// TIA Portal V20 export
FUNCTION_BLOCK "LER_GantryHoming"   // FB103, LAD
// stored: Access Published, MemoryReserve 100, SetENOAutomatically false
   VAR_INPUT
      enableManualCmds { ExternalAccessible := 'False'; ExternalVisible := 'False'; ExternalWritable := 'False'} : Bool;
      startConidition { ExternalAccessible := 'False'; ExternalVisible := 'False'; ExternalWritable := 'False'} : Bool := false;
      insync { ExternalAccessible := 'False'; ExternalVisible := 'False'; ExternalWritable := 'False'} : Bool;
      masterControlNode { ExternalAccessible := 'False'; ExternalVisible := 'False'; ExternalWritable := 'False'} : "LBC_typeAxis64PosControlNodeMonitoring";
      slaveControlNode { ExternalAccessible := 'False'; ExternalVisible := 'False'; ExternalWritable := 'False'} : "LBC_typeAxis64PosControlNodeMonitoring";
   END_VAR
   VAR_OUTPUT
      resetRequest { ExternalAccessible := 'False'; ExternalVisible := 'False'; ExternalWritable := 'False'} : Bool;
      homingRequest { ExternalAccessible := 'False'; ExternalVisible := 'False'; ExternalWritable := 'False'} : Bool;
      gearInRequest { ExternalAccessible := 'False'; ExternalVisible := 'False'; ExternalWritable := 'False'} : Bool;
      busy { ExternalAccessible := 'False'; ExternalVisible := 'False'; ExternalWritable := 'False'} : Bool;
      done { ExternalAccessible := 'False'; ExternalVisible := 'False'; ExternalWritable := 'False'} : Bool;
   END_VAR
   VAR
      statStep { ExternalAccessible := 'False'; ExternalVisible := 'False'; ExternalWritable := 'False'} : DInt;
      statLocalBit { ExternalAccessible := 'False'; ExternalVisible := 'False'; ExternalWritable := 'False'} : Array[0..99] of Bool;
      statTonTime { ExternalAccessible := 'False'; ExternalVisible := 'False'; ExternalWritable := 'False'} : Array[0..99] of TON_TIME;
   END_VAR
   VAR_TEMP   // added for the SCL form of the ladder/FBD networks
      _w1 : Bool;
   END_VAR
BEGIN

REGION Network 1: STEP[0] : Start Condition
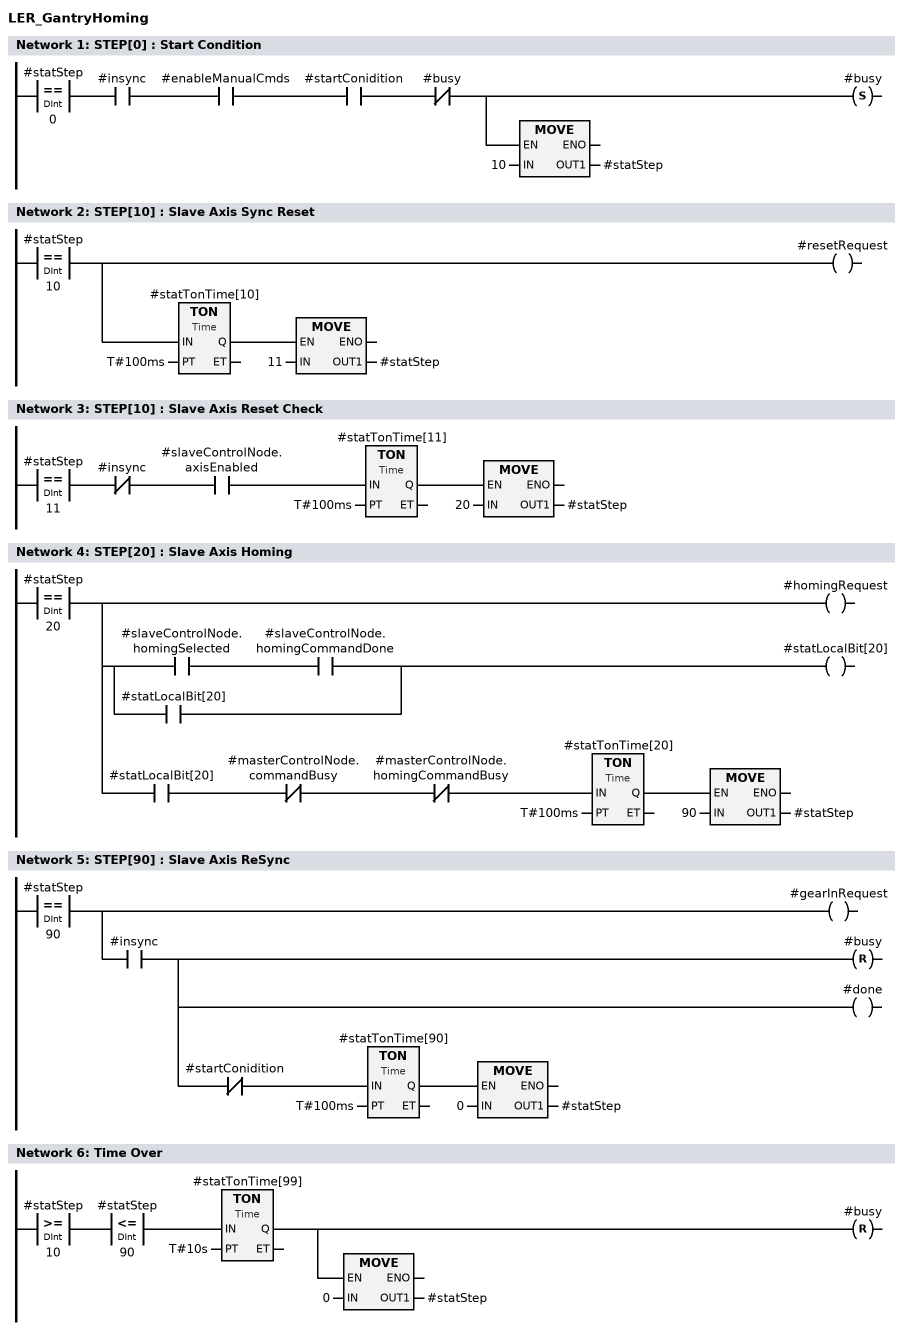
   RUNG wire#powerrail
      { S7_Templates := "SrcType := DInt" } EQ_Contact(in1 := #statStep, in2 := 0)
      Contact( #insync )
      Contact( #enableManualCmds )
      Contact( #startConidition )
      I_Contact( #busy )
      wire#w1
      S_Coil( #busy )
   END_RUNG
   RUNG wire#w1
      Move(in := 10, out1 => #statStep)
   END_RUNG
   // the same network as SCL:
   #_w1 := (#statStep = 0) AND #insync AND #enableManualCmds AND #startConidition AND NOT #busy;
   IF #_w1 THEN
       #busy := TRUE;
       #statStep := 10;
   END_IF;
END_REGION

REGION Network 2: STEP[10] : Slave Axis Sync Reset
   RUNG wire#powerrail
      { S7_Templates := "SrcType := DInt" } EQ_Contact(in1 := #statStep, in2 := 10)
      wire#w1
      Coil( #resetRequest )
   END_RUNG
   RUNG wire#w1
      { S7_Templates := "time_type := Time" } #statTonTime[10].TON(pt := T#100ms, et =>)
      Move(in := 11, out1 => #statStep)
   END_RUNG
   // the same network as SCL:
   #resetRequest := #statStep = 10;
   #statTonTime[10].TON(IN := #resetRequest, PT := T#100ms);
   IF #statTonTime[10].Q THEN #statStep := 11; END_IF;
END_REGION

REGION Network 3: STEP[10] : Slave Axis Reset Check
   RUNG wire#powerrail
      { S7_Templates := "SrcType := DInt" } EQ_Contact(in1 := #statStep, in2 := 11)
      I_Contact( #insync )
      Contact( #slaveControlNode.axisEnabled )
      { S7_Templates := "time_type := Time" } #statTonTime[11].TON(pt := T#100ms, et =>)
      Move(in := 20, out1 => #statStep)
   END_RUNG
   // the same network as SCL:
   #statTonTime[11].TON(IN := (#statStep = 11) AND NOT #insync AND #slaveControlNode.axisEnabled, PT := T#100ms);
   IF #statTonTime[11].Q THEN #statStep := 20; END_IF;
END_REGION

REGION Network 4: STEP[20] : Slave Axis Homing
   RUNG wire#powerrail
      { S7_Templates := "SrcType := DInt" } EQ_Contact(in1 := #statStep, in2 := 20)
      wire#w1
      Coil( #homingRequest )
   END_RUNG
   RUNG wire#w1
      Contact( #slaveControlNode.homingSelected )
      Contact( #slaveControlNode.homingCommandDone )
      wire#w2
      Coil( #statLocalBit[20] )
   END_RUNG
   RUNG wire#w1
      Contact( #statLocalBit[20] )
   END_RUNG wire#w2
   RUNG wire#w1
      Contact( #statLocalBit[20] )
      I_Contact( #masterControlNode.commandBusy )
      I_Contact( #masterControlNode.homingCommandBusy )
      { S7_Templates := "time_type := Time" } #statTonTime[20].TON(pt := T#100ms, et =>)
      Move(in := 90, out1 => #statStep)
   END_RUNG
   // the same network as SCL:
   #homingRequest := #statStep = 20;
   #statLocalBit[20] := #homingRequest AND ((#slaveControlNode.homingSelected AND #slaveControlNode.homingCommandDone) OR #statLocalBit[20]);
   #statTonTime[20].TON(IN := #homingRequest AND #statLocalBit[20] AND NOT #masterControlNode.commandBusy AND NOT #masterControlNode.homingCommandBusy,
                        PT := T#100ms);
   IF #statTonTime[20].Q THEN #statStep := 90; END_IF;
END_REGION

REGION Network 5: STEP[90] : Slave Axis ReSync
   RUNG wire#powerrail
      { S7_Templates := "SrcType := DInt" } EQ_Contact(in1 := #statStep, in2 := 90)
      wire#w1
      Coil( #gearInRequest )
   END_RUNG
   RUNG wire#w1
      Contact( #insync )
      wire#w2
      R_Coil( #busy )
   END_RUNG
   RUNG wire#w2
      Coil( #done )
   END_RUNG
   RUNG wire#w2
      I_Contact( #startConidition )
      { S7_Templates := "time_type := Time" } #statTonTime[90].TON(pt := T#100ms, et =>)
      Move(in := 0, out1 => #statStep)
   END_RUNG
   // the same network as SCL:
   #gearInRequest := #statStep = 90;
   #_w1 := #gearInRequest AND #insync;
   IF #_w1 THEN #busy := FALSE; END_IF;
   #done := #_w1;
   #statTonTime[90].TON(IN := #_w1 AND NOT #startConidition, PT := T#100ms);
   IF #statTonTime[90].Q THEN #statStep := 0; END_IF;
END_REGION

REGION Network 6: Time Over
   RUNG wire#powerrail
      { S7_Templates := "SrcType := DInt" } GE_Contact(in1 := #statStep, in2 := 10)
      { S7_Templates := "SrcType := DInt" } LE_Contact(in1 := #statStep, in2 := 90)
      { S7_Templates := "time_type := Time" } #statTonTime[99].TON(pt := T#10s, et =>)
      wire#w1
      R_Coil( #busy )
   END_RUNG
   RUNG wire#w1
      Move(in := 0, out1 => #statStep)
   END_RUNG
   // the same network as SCL:
   #statTonTime[99].TON(IN := (#statStep >= 10) AND (#statStep <= 90), PT := T#10s);
   IF #statTonTime[99].Q THEN
       #busy := FALSE;
       #statStep := 0;
   END_IF;
END_REGION
END_FUNCTION_BLOCK
